RoboDK station: plane_optimization.rdk

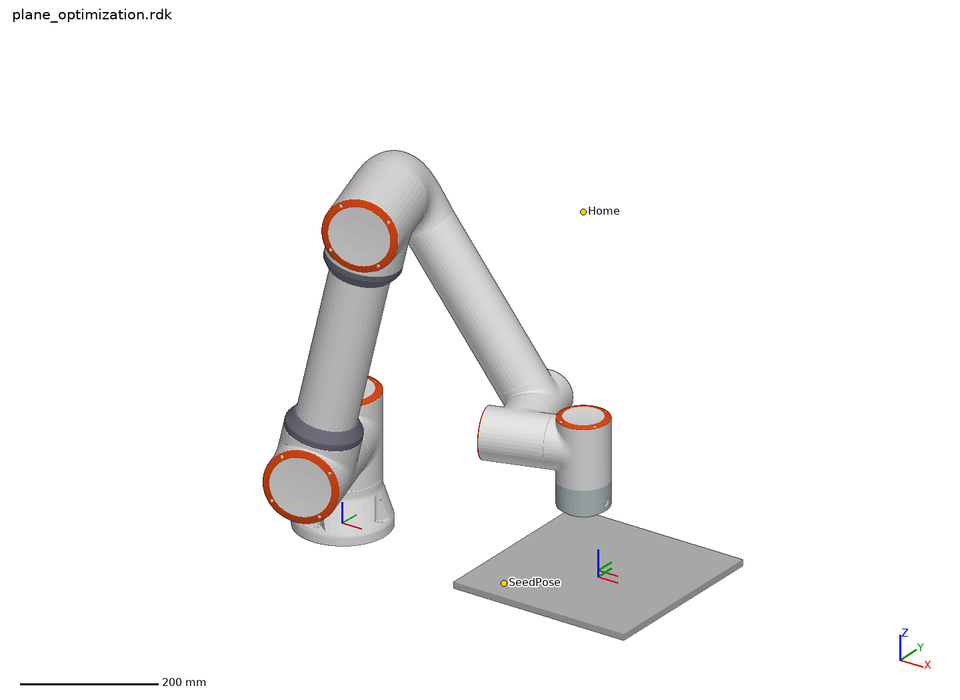
[picture v0: the station drawn from its stored meshes, robots at their saved joint values, targets as dots, program paths as lines]
Station plane_optimization (saved by RoboDK 6.0.4). Poses are relative to the parent item; angles as X-Y-Z fixed-axis rotations.
  - frame FAIRINO FR5 Base at (0, 0, 0) mm
    - robot FAIRINO FR5: 6 axes
        modified DH rows (alpha deg, a mm, theta deg, d mm): 0, 0, 0, 152; 90, 0, 180, 0; 0, 425, 0, 0; 0, 395, 0, 102; -90, 0, 0, 102; 90, 0, 180, 100
        joint limits [-175, -265, -160, -265, -175, -175] to [175, 85, 160, 85, 175, 175]; home [0, -90, -90, 0, 90, 0]; saved at [17.556, -102.09, -136.627, -31.283, 90, 17.556]
      - tool Tool 1, TCP at (0, 0, 80) mm
  - frame PlateFrame at (450, 0, 50) mm
    - target Home (Cartesian target) at (45, -102, 629) mm, rotated rx -90 ry 0 rz -90 deg; joints [0, -90, -90, 0, 90, 0] of FAIRINO FR5
    - target SeedPose (Cartesian target) at (-86.41, -113.01, 0) mm, rotated rx -180 ry 0 rz -90 deg; joints [-1.727, -99.033, -140.866, -30.102, 90, -1.727] of FAIRINO FR5
  - frame Frame 3 at (450, 0, 40) mm
    - object plane at (0, 0, 0) mm, size 300 x 300 x 10 mm, geometry from plane.stl
